FUNCTION_BLOCK RateLimiter (* Composite Function Block Type *)
  (* Standard: 61499-2 *)
  (* Version 0.0, 2018-09-25, 4DIAC-IDE, 4DIAC-Consortium *)
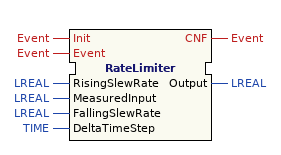
  EVENT_INPUT
    Init; (* Normal Execution Request *)
    Event;
  END_EVENT
  EVENT_OUTPUT
    CNF; (* Execution Confirmation *)
  END_EVENT
  VAR_INPUT
    RisingSlewRate : LREAL;
    MeasuredInput : LREAL;
    FallingSlewRate : LREAL;
    DeltaTimeStep : TIME;
  END_VAR
  VAR_OUTPUT
    Output : LREAL;
  END_VAR
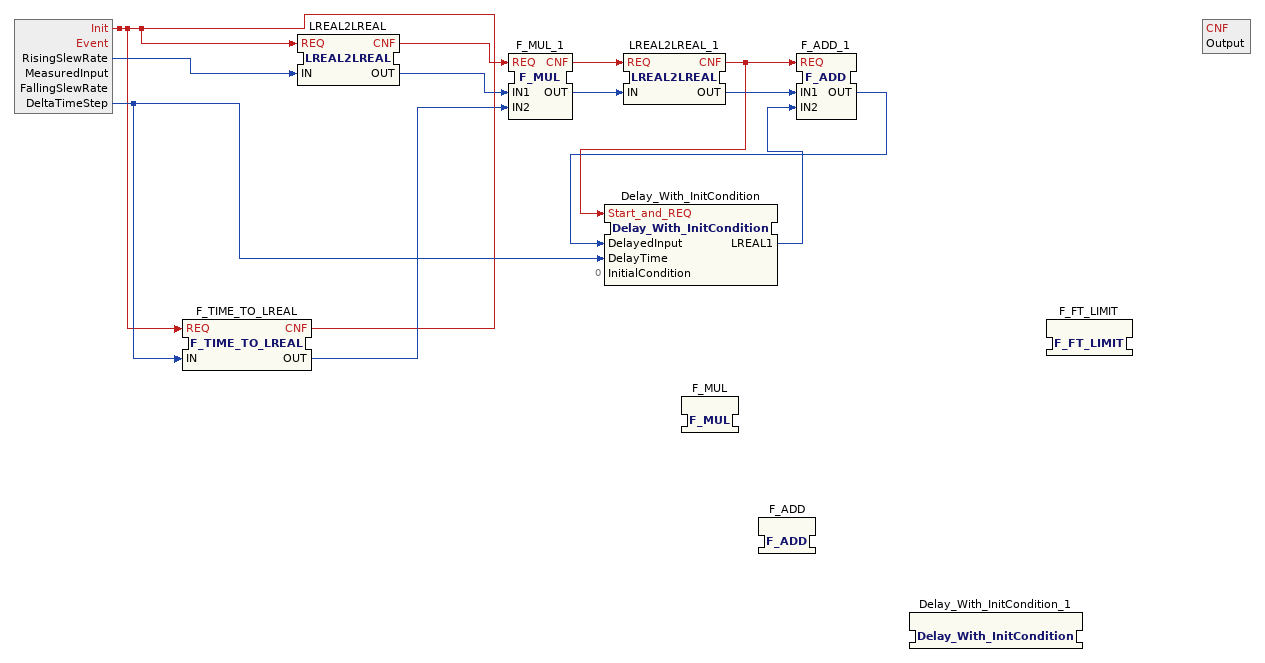
  FBS
    F_TIME_TO_LREAL : F_TIME_TO_LREAL;
    F_FT_LIMIT : F_FT_LIMIT;
    F_MUL : F_MUL;
    F_MUL_1 : F_MUL;
    LREAL2LREAL : LREAL2LREAL;
    LREAL2LREAL_1 : LREAL2LREAL;
    Delay_With_InitCondition : Delay_With_InitCondition(InitialCondition := 0);
    Delay_With_InitCondition_1 : Delay_With_InitCondition;
    F_ADD : F_ADD;
    F_ADD_1 : F_ADD;
  END_FBS
  EVENT_CONNECTIONS
    Init TO F_TIME_TO_LREAL.REQ;
    Init TO F_MUL_1.REQ;
    Init TO LREAL2LREAL.REQ;
    LREAL2LREAL.CNF TO F_MUL_1.REQ;
    F_MUL_1.CNF TO LREAL2LREAL_1.REQ;
    LREAL2LREAL_1.CNF TO F_ADD_1.REQ;
    F_TIME_TO_LREAL.CNF TO F_MUL_1.REQ;
    LREAL2LREAL_1.CNF TO Delay_With_InitCondition.Start_and_REQ;
  END_CONNECTIONS
  DATA_CONNECTIONS
    DeltaTimeStep TO F_TIME_TO_LREAL.IN;
    RisingSlewRate TO LREAL2LREAL.IN;
    LREAL2LREAL.OUT TO F_MUL_1.IN1;
    F_MUL_1.OUT TO LREAL2LREAL_1.IN;
    LREAL2LREAL_1.OUT TO F_ADD_1.IN1;
    F_TIME_TO_LREAL.OUT TO F_MUL_1.IN2;
    Delay_With_InitCondition.LREAL1 TO F_ADD_1.IN2;
    F_ADD_1.OUT TO Delay_With_InitCondition.DelayedInput;
    DeltaTimeStep TO Delay_With_InitCondition.DelayTime;
  END_CONNECTIONS
END_FUNCTION_BLOCK
